% RSLogix 500 project filling_station_v2.RSS, saved by version 8.30.00.16 %
PROJECT "UNTITLED"    % processor: Bul.1763 MicroLogix 1100 Series B %

PROGRAM FILES
  LAD 2   3 rungs
  LAD 3 "IO"  10 rungs
  LAD 4 "CONTROLS"  12 rungs

DATA FILES
  O0 OUTPUT  4 elements
  I1 INPUT  6 elements
  S2 STATUS  66 elements
  B3 BINARY  4 elements
  T4 TIMER  1 elements
  C5 COUNTER  1 elements
  R6 CONTROL  1 elements
  N7 INTEGER  10 elements
  F8 FLOAT  1 elements

LADDER 2
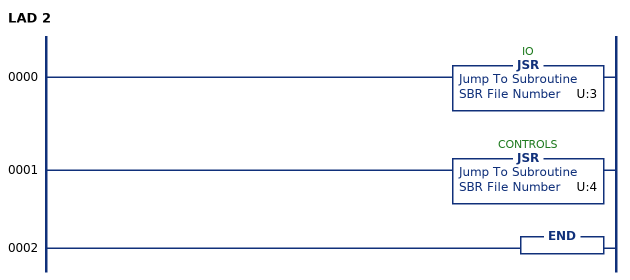
% Rung: 0 %
SOR JSR U:3 EOR
%   U:3  "IO" %
% Rung: 1 %
SOR JSR U:4 EOR
%   U:4  "CONTROLS" %
% Rung: 2 %
SOR END EOR

LADDER 3 "IO"
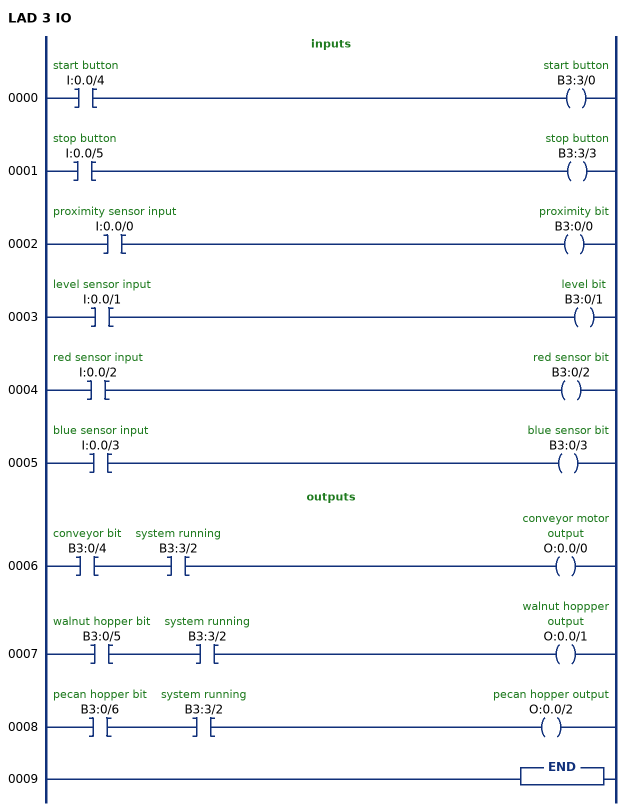
% Rung: 0 %
% TITLE: inputs %
SOR XIC I:0.0/4 OTE B3:3/0 EOR
%   I:0.0/4  "start button" %
%   B3:3/0  "start button" %
% Rung: 1 %
SOR XIC I:0.0/5 OTE B3:3/3 EOR
%   I:0.0/5  "stop button" %
%   B3:3/3  "stop button" %
% Rung: 2 %
SOR XIC I:0.0/0 OTE B3:0/0 EOR
%   I:0.0/0  "proximity sensor input" %
%   B3:0/0  "proximity bit" %
% Rung: 3 %
SOR XIC I:0.0/1 OTE B3:0/1 EOR
%   I:0.0/1  "level sensor input" %
%   B3:0/1  "level bit" %
% Rung: 4 %
SOR XIC I:0.0/2 OTE B3:0/2 EOR
%   I:0.0/2  "red sensor input" %
%   B3:0/2  "red sensor bit" %
% Rung: 5 %
SOR XIC I:0.0/3 OTE B3:0/3 EOR
%   I:0.0/3  "blue sensor input" %
%   B3:0/3  "blue sensor bit" %
% Rung: 6 %
% TITLE: outputs %
SOR XIC B3:0/4 XIC B3:3/2 OTE O:0.0/0 EOR
%   B3:0/4  "conveyor bit" %
%   B3:3/2  "system running" %
%   O:0.0/0  "conveyor motor output" %
% Rung: 7 %
SOR XIC B3:0/5 XIC B3:3/2 OTE O:0.0/1 EOR
%   B3:0/5  "walnut hopper bit" %
%   B3:3/2  "system running" %
%   O:0.0/1  "walnut hoppper output" %
% Rung: 8 %
SOR XIC B3:0/6 XIC B3:3/2 OTE O:0.0/2 EOR
%   B3:0/6  "pecan hopper bit" %
%   B3:3/2  "system running" %
%   O:0.0/2  "pecan hopper output" %
% Rung: 9 %
SOR END EOR

LADDER 4 "CONTROLS"
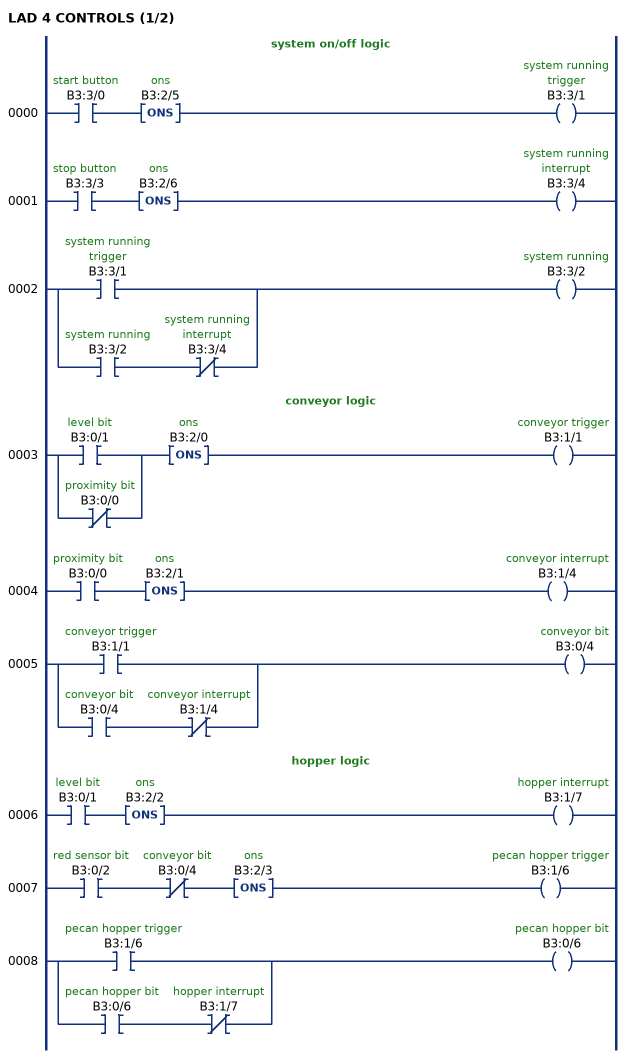
% Rung: 0 %
% TITLE: system on/off logic %
SOR XIC B3:3/0 ONS B3:2/5 OTE B3:3/1 EOR
%   B3:3/0  "start button" %
%   B3:2/5  "ons" %
%   B3:3/1  "system running trigger" %
% Rung: 1 %
SOR XIC B3:3/3 ONS B3:2/6 OTE B3:3/4 EOR
%   B3:3/3  "stop button" %
%   B3:2/6  "ons" %
%   B3:3/4  "system running interrupt" %
% Rung: 2 %
SOR BST XIC B3:3/1 NXB XIC B3:3/2 XIO B3:3/4 BND OTE B3:3/2 EOR
%   B3:3/1  "system running trigger" %
%   B3:3/2  "system running" %
%   B3:3/4  "system running interrupt" %
% Rung: 3 %
% TITLE: conveyor logic %
SOR BST XIC B3:0/1 NXB XIO B3:0/0 BND ONS B3:2/0 OTE B3:1/1 EOR
%   B3:0/1  "level bit" %
%   B3:0/0  "proximity bit" %
%   B3:2/0  "ons" %
%   B3:1/1  "conveyor trigger" %
% Rung: 4 %
SOR XIC B3:0/0 ONS B3:2/1 OTE B3:1/4 EOR
%   B3:0/0  "proximity bit" %
%   B3:2/1  "ons" %
%   B3:1/4  "conveyor interrupt" %
% Rung: 5 %
SOR BST XIC B3:1/1 NXB XIC B3:0/4 XIO B3:1/4 BND OTE B3:0/4 EOR
%   B3:1/1  "conveyor trigger" %
%   B3:0/4  "conveyor bit" %
%   B3:1/4  "conveyor interrupt" %
% Rung: 6 %
% TITLE: hopper logic %
SOR XIC B3:0/1 ONS B3:2/2 OTE B3:1/7 EOR
%   B3:0/1  "level bit" %
%   B3:2/2  "ons" %
%   B3:1/7  "hopper interrupt" %
% Rung: 7 %
SOR XIC B3:0/2 XIO B3:0/4 ONS B3:2/3 OTE B3:1/6 EOR
%   B3:0/2  "red sensor bit" %
%   B3:0/4  "conveyor bit" %
%   B3:2/3  "ons" %
%   B3:1/6  "pecan hopper trigger" %
% Rung: 8 %
SOR BST XIC B3:1/6 NXB XIC B3:0/6 XIO B3:1/7 BND OTE B3:0/6 EOR
%   B3:1/6  "pecan hopper trigger" %
%   B3:0/6  "pecan hopper bit" %
%   B3:1/7  "hopper interrupt" %

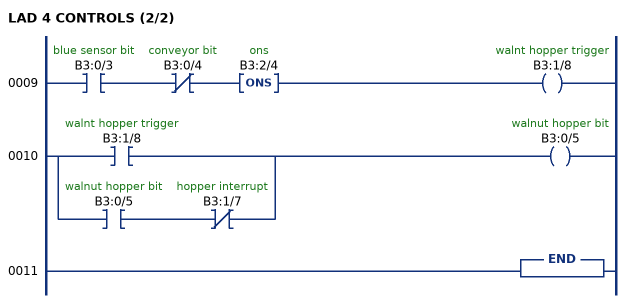
% Rung: 9 %
SOR XIC B3:0/3 XIO B3:0/4 ONS B3:2/4 OTE B3:1/8 EOR
%   B3:0/3  "blue sensor bit" %
%   B3:0/4  "conveyor bit" %
%   B3:2/4  "ons" %
%   B3:1/8  "walnt hopper trigger" %
% Rung: 10 %
SOR BST XIC B3:1/8 NXB XIC B3:0/5 XIO B3:1/7 BND OTE B3:0/5 EOR
%   B3:1/8  "walnt hopper trigger" %
%   B3:0/5  "walnut hopper bit" %
%   B3:1/7  "hopper interrupt" %
% Rung: 11 %
SOR END EOR

OTHER DOCUMENTED ADDRESSES
  B3:0/7  "ons"
  B3:0/8  "conveyor trigger"
  B3:0/9  "ons"
  B3:0/10  "conveyor trigger interrupt"
  B3:0/11  "ons"
  B3:0/12  "ons"
  B3:0/13  "ons"
  B3:0/14  "pecan trigger"
  B3:0/15  "walnut trigger"
  B3:1/0  "ons"
  B3:1/2  "ons"
  B3:1/3  "ons"
  B3:1/5  "ons"
  B3:1/9  "ons"
  N7:0  "conveyor state: 0 = stopped 1 = moving"
  N7:0/0  "conveyor state: 0 = stopped 1 = moving"
  N7:0/1  "conveyor state: zero"
  N7:1  "hopper state: 0 = off 1 = pack pecan 2 = pack walnut"
  U:5  "CONTROLS"
  U:6  "CONTROLS"

COMMENTS NOT ATTACHED TO A CURRENT RUNG
  B3:0/14: packing logic
  B3:1/3: inputs

DATA TABLE (non-zero values as saved)
DATA B3
% B3:0 % 0X0201 0X0000 0X0000 0X0000
